FUNCTION_BLOCK FB_AnalogueInputTest
VAR_INPUT
END_VAR
VAR_OUTPUT
END_VAR
VAR
	analogueIn : AnalogueStatus;
	fbAnalogue : FB_AnalogueInputBase(SignalType := SignalType._0_20mA, Resolution := Resolution._12Bit, ProceesData := analogueIn);
END_VAR

METHOD CheckConvertedValue : BOOL
VAR_INPUT
END_VAR
END_METHOD

METHOD CheckError : BOOL
VAR_INPUT
END_VAR
END_METHOD

METHOD CheckRawValue : BOOL
VAR_INPUT
END_VAR
END_METHOD

END_FUNCTION_BLOCK

(* stored: Version 1.1.0.1, ProductVersion 3.1.4024.5
   POU FB_AnalogueInputTest: Id {4b624b13-8320-4357-a153-692da183e6e0}, SpecialFunc None
   Method CheckConvertedValue: Id {1d8e5d28-cc2c-40d8-8717-72a573ebe234}
   Method CheckError: Id {a96aba15-f2f0-4b1b-bddc-ae4a79e277df}
   Method CheckRawValue: Id {d4ed59de-963f-483a-94ed-421617e5b806} *)
